FUNCTION_BLOCK FB_Bel_RGBW
VAR_INPUT
	Freigabe_auto			: BOOL;
	Freigabe_Deakt_auto		: BOOL;
	Betrieb_Anford_auto		: BOOL;
	Farbcode			: STRING;
	Adresse_R				: BYTE;
	Adresse_G				: BYTE;
	Adresse_B				: BYTE;
	Adresse_W				: BYTE;
	Quittierung				: BOOL;
	AdressType				: E_DALIV2AddrType;
	Reset					: BOOL;

END_VAR
VAR_OUTPUT
	{attribute 'OPC.UA.DA' := '1'}Steuerung				: ST_Bel_Steuerung;		
	{attribute 'OPC.UA.DA' := '1'}Stellwert				: ST_Bel_Stellwert;		
	{attribute 'OPC.UA.DA' := '1'}Zustand					: ST_Bel_Zustand;	
	{attribute 'OPC.UA.DA' := '1'}Parameter				: ST_Bel_Parameter;		
END_VAR
VAR
	Beleuchtung_R			: FB_Bel_Einzel_farbe;
	Beleuchtung_G			: FB_Bel_Einzel_farbe;
	Beleuchtung_B			: FB_Bel_Einzel_farbe;
	Beleuchtung_W			: FB_Bel_Einzel_farbe;

	Stellwert_R_Regelung	: REAL;
	Stellwert_G_Regelung	: REAL;
	Stellwert_B_Regelung	: REAL;
	Stellwert_W_Regelung	: REAL;

	Zustand_Bel_R			: ST_BEL_Zustand;
	Zustand_Bel_G			: ST_BEL_Zustand;
	Zustand_Bel_B			: ST_BEL_Zustand;
	Zustand_Bel_W			: ST_BEL_Zustand;

	Logik					: FB_Bel_RGBW_Logik;
	Ablaufsteuerung			: FB_Bel_RGBW_Ablaufsteuerung;

	Regelung				: FB_Bel_RGBW_Regelung;
	QuitTrig				: FB_SetResetFallTrigger;
	Anschaltung				: BOOL;

	Time_on: TON;
	Reset1: TON;
END_VAR
VAR // added by the converter: edge detectors and wires of the graphical bodies
    _w1 : ANY;
END_VAR

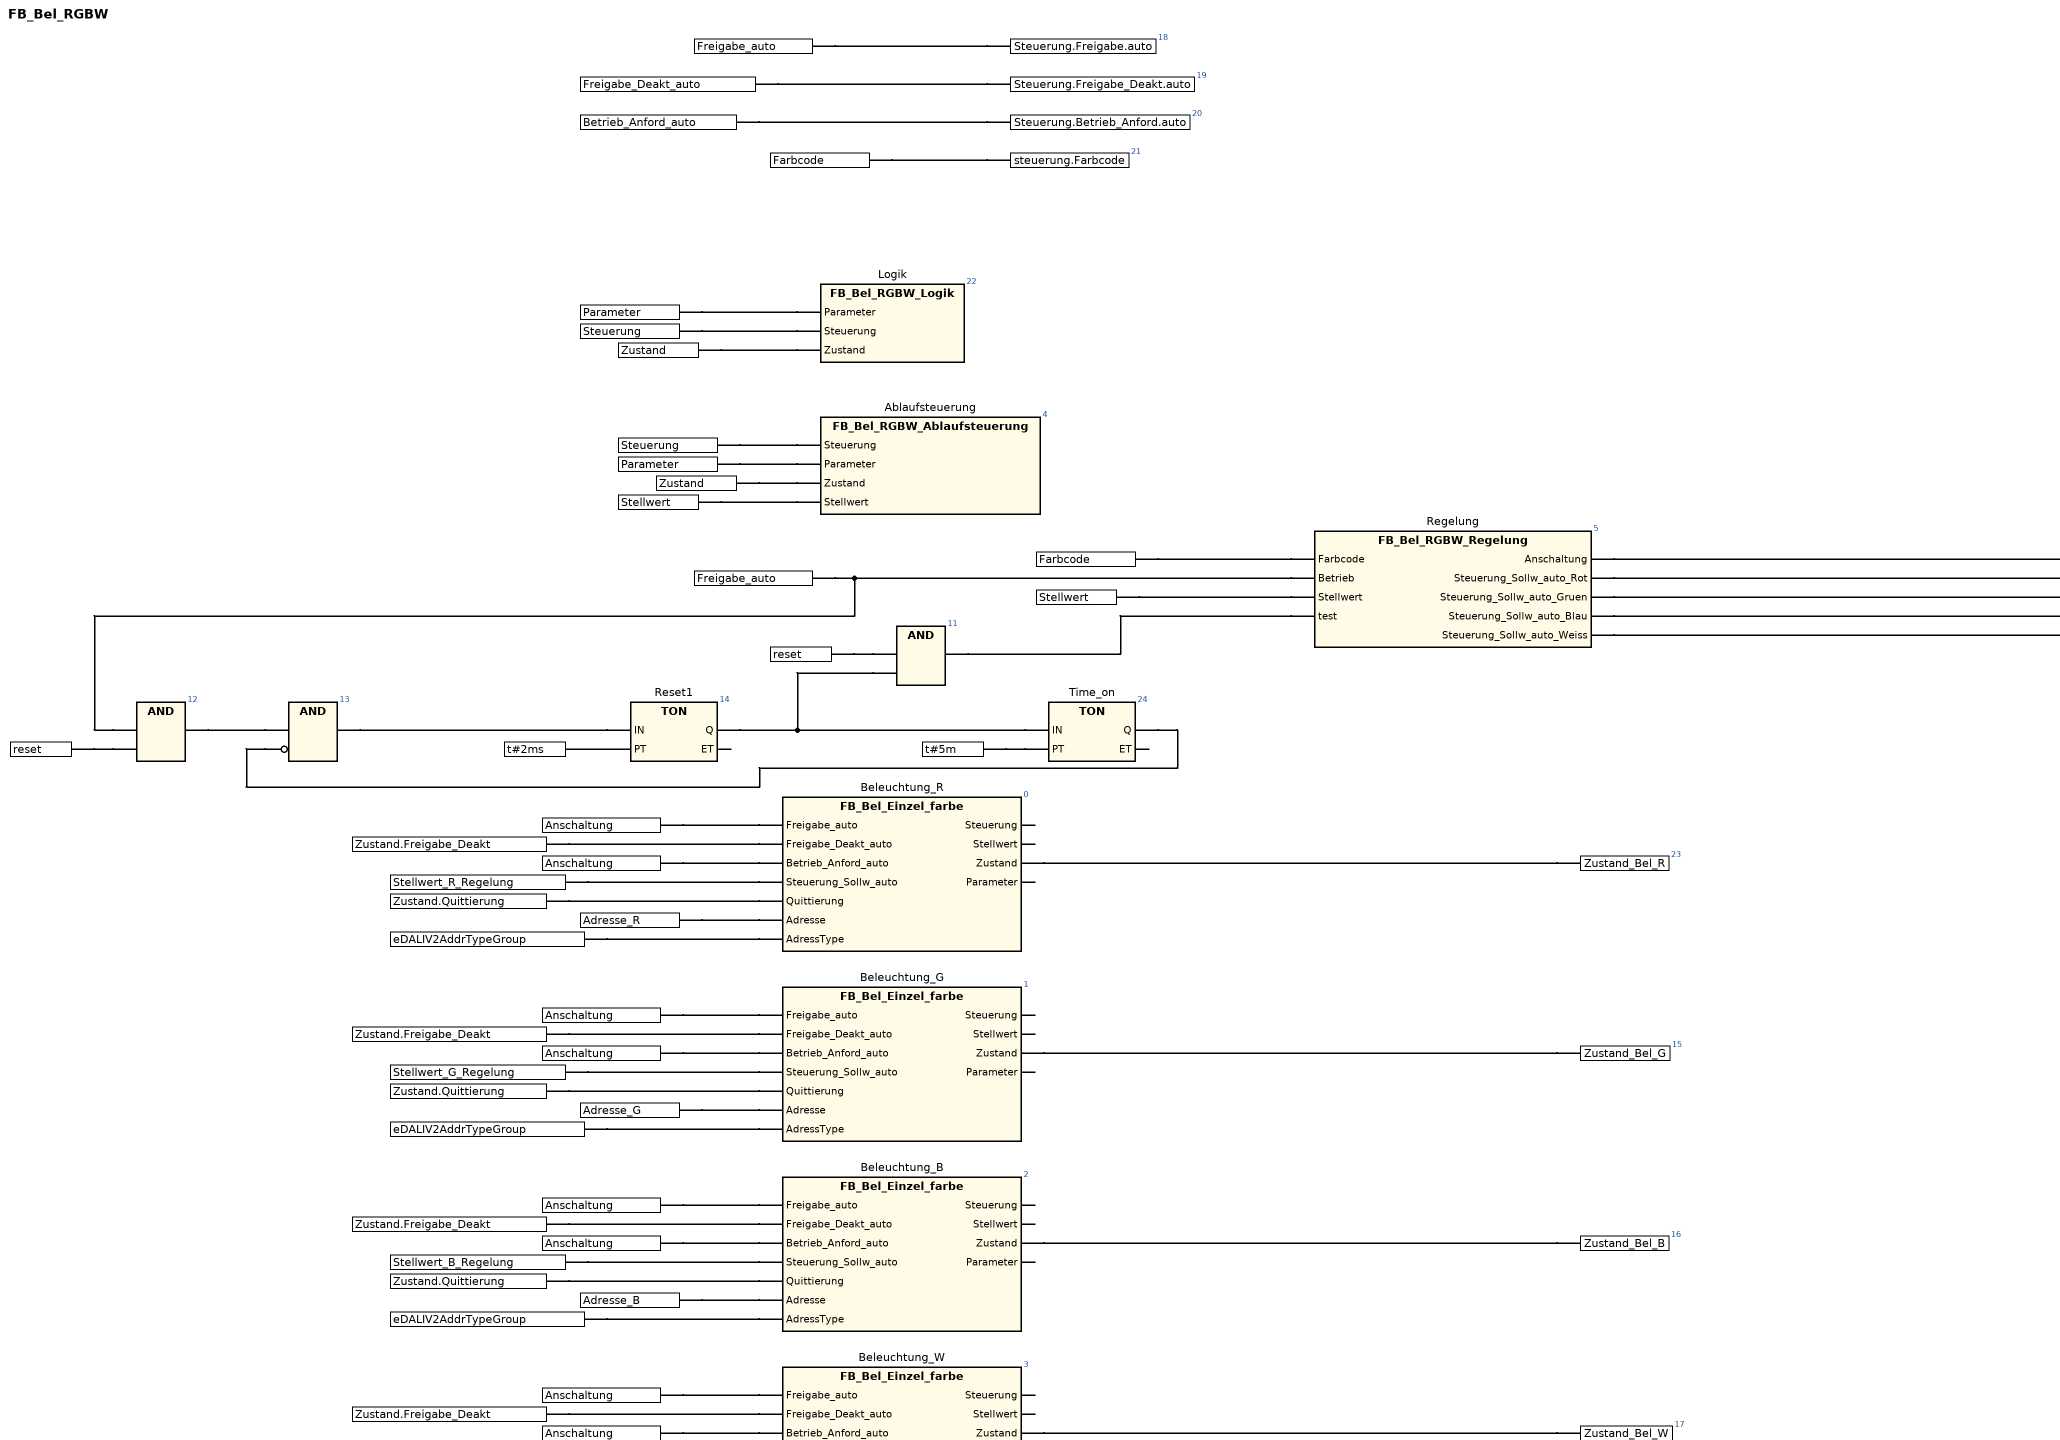
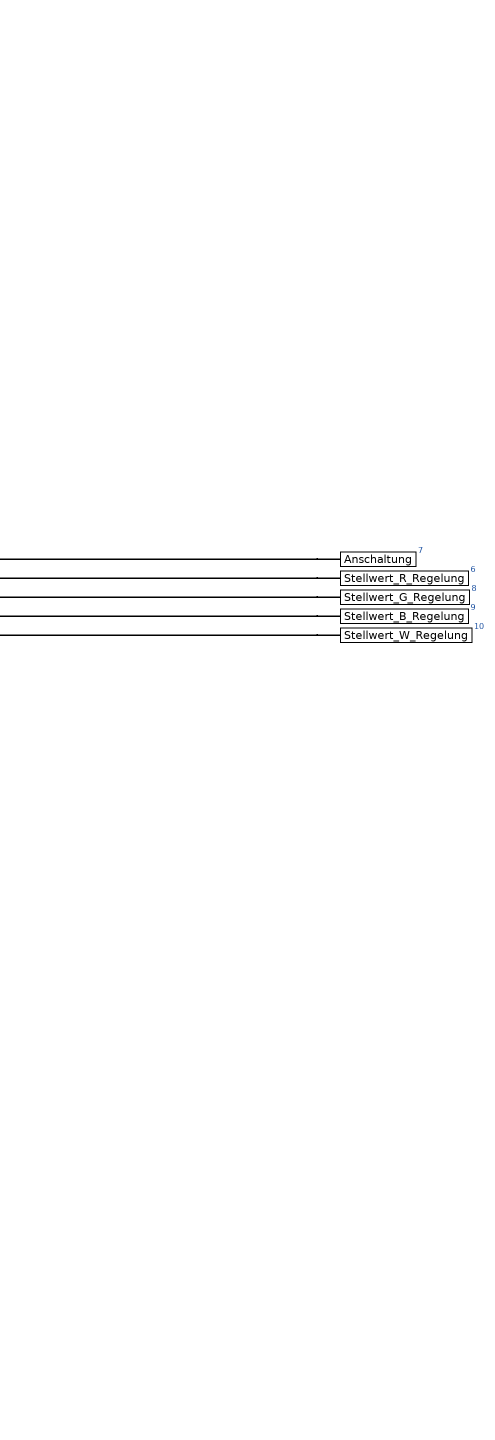
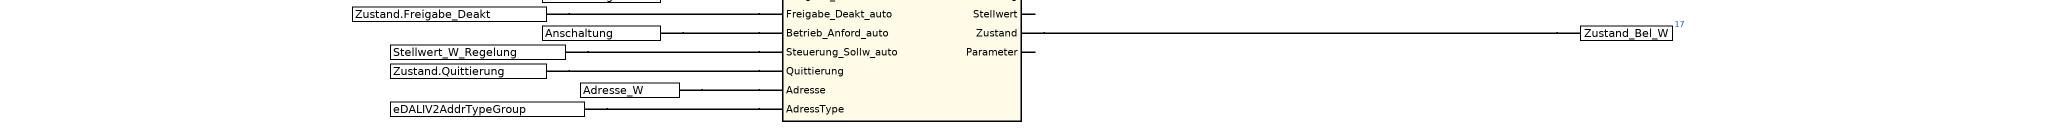
Beleuchtung_R(
    Freigabe_auto := Anschaltung,
    Freigabe_Deakt_auto := Zustand.Freigabe_Deakt,
    Betrieb_Anford_auto := Anschaltung,
    Steuerung_Sollw_auto := Stellwert_R_Regelung,
    Quittierung := Zustand.Quittierung,
    Adresse := Adresse_R,
    AdressType := eDALIV2AddrTypeGroup); // FB_Bel_Einzel_farbe
Beleuchtung_G(
    Freigabe_auto := Anschaltung,
    Freigabe_Deakt_auto := Zustand.Freigabe_Deakt,
    Betrieb_Anford_auto := Anschaltung,
    Steuerung_Sollw_auto := Stellwert_G_Regelung,
    Quittierung := Zustand.Quittierung,
    Adresse := Adresse_G,
    AdressType := eDALIV2AddrTypeGroup); // FB_Bel_Einzel_farbe
Beleuchtung_B(
    Freigabe_auto := Anschaltung,
    Freigabe_Deakt_auto := Zustand.Freigabe_Deakt,
    Betrieb_Anford_auto := Anschaltung,
    Steuerung_Sollw_auto := Stellwert_B_Regelung,
    Quittierung := Zustand.Quittierung,
    Adresse := Adresse_B,
    AdressType := eDALIV2AddrTypeGroup); // FB_Bel_Einzel_farbe
Beleuchtung_W(
    Freigabe_auto := Anschaltung,
    Freigabe_Deakt_auto := Zustand.Freigabe_Deakt,
    Betrieb_Anford_auto := Anschaltung,
    Steuerung_Sollw_auto := Stellwert_W_Regelung,
    Quittierung := Zustand.Quittierung,
    Adresse := Adresse_W,
    AdressType := eDALIV2AddrTypeGroup); // FB_Bel_Einzel_farbe
Ablaufsteuerung(Steuerung := Steuerung, Parameter := Parameter, Zustand := Zustand, Stellwert := Stellwert); // FB_Bel_RGBW_Ablaufsteuerung
Regelung(Farbcode := Farbcode, Betrieb := Freigabe_auto, Stellwert := Stellwert, test := _w1); // FB_Bel_RGBW_Regelung
Stellwert_R_Regelung := Regelung.Steuerung_Sollw_auto_Rot;
Anschaltung := Regelung.Anschaltung;
Stellwert_G_Regelung := Regelung.Steuerung_Sollw_auto_Gruen;
Stellwert_B_Regelung := Regelung.Steuerung_Sollw_auto_Blau;
Stellwert_W_Regelung := Regelung.Steuerung_Sollw_auto_Weiss;
_w1 := reset AND Reset1.Q;
Reset1(IN := (Freigabe_auto AND reset) AND NOT Time_on.Q, PT := t#2ms); // TON
Zustand_Bel_G := Beleuchtung_G.Zustand;
Zustand_Bel_B := Beleuchtung_B.Zustand;
Zustand_Bel_W := Beleuchtung_W.Zustand;
Steuerung.Freigabe.auto := Freigabe_auto;
Steuerung.Freigabe_Deakt.auto := Freigabe_Deakt_auto;
Steuerung.Betrieb_Anford.auto := Betrieb_Anford_auto;
steuerung.Farbcode := Farbcode;
Logik(Parameter := Parameter, Steuerung := Steuerung, Zustand := Zustand); // FB_Bel_RGBW_Logik
Zustand_Bel_R := Beleuchtung_R.Zustand;
Time_on(IN := Reset1.Q, PT := t#5m); // TON

END_FUNCTION_BLOCK

(* stored: Version 1.1.0.1, ProductVersion 3.1.4024.10
   POU FB_Bel_RGBW: Id {2fddff3f-9dd2-4ac8-9bdb-308221aa9669}, SpecialFunc None *)
